RoboDK station: Sheet A.rdk

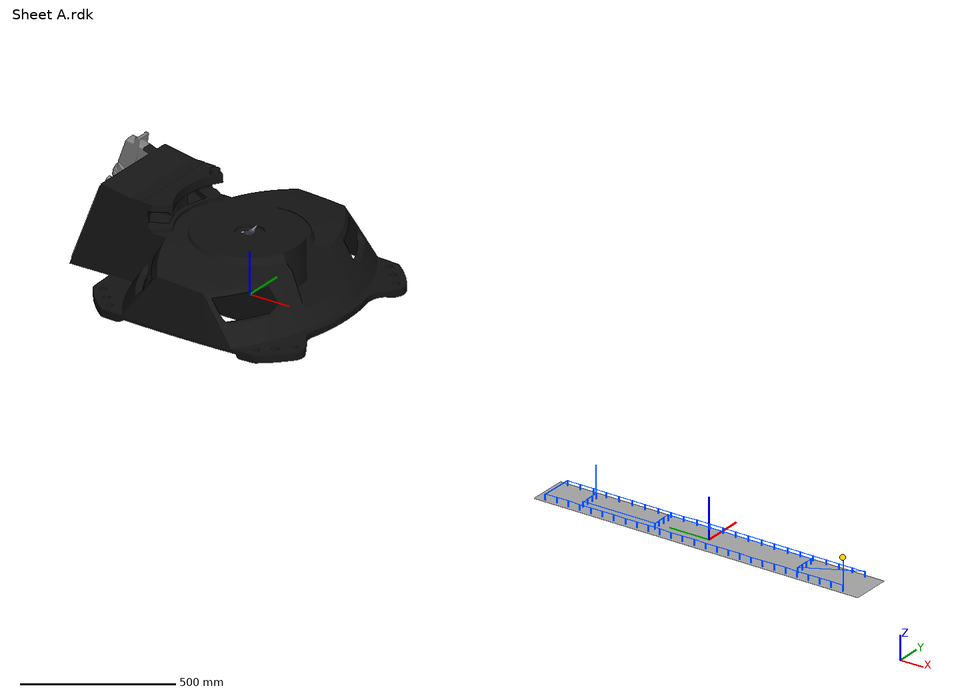
[picture v0: the station drawn from its stored meshes, robots at their saved joint values, targets as dots, program paths as lines]
Station Sheet A (saved by RoboDK 5.2.3). Poses are relative to the parent item; angles as X-Y-Z fixed-axis rotations.
  - frame KUKA KR 210 R2700 extra Base at (0, 0, 0) mm
    - robot KUKA KR 210 R2700 extra: 6 axes, payload 210 kg, reach 2696 mm, repeatability 0.06 mm, weight 1068 kg
        joint limits [-185, -140, -120, -350, -125, -350] to [185, -5, 155, 350, 125, 350]; home [0, -90, 90, 0, 0, 0]; saved at [-1.926, -24.263, 90.653, -184.563, 15.421, 182.902]
      - tool Spindle, TCP at (32, 0, 260) mm, rotated rx 0 ry 39 rz 0 deg, size 157.3 x 72 x 259.9 mm
  - frame Frame 2 at (1800, 0, -372.68) mm, rotated rx 0 ry 0 rz 90 deg
    - object Sheet A stp at (0, 0, 0) mm, size 148.8 x 1269.1 x 0.8 mm, geometry from Sheet A stp.stp
    - object Sheet A-box 1 Hole positioning at (0, 0, 0) mm, 63 curves, geometry from Point 63
  - machining project Point settings: rotZ(0) | rotX(0)*rotY(0) | rotZ(0) | onStart | onPathStart | onApproach | onPoint | onRetract | onFinish | SetRPM(%1) | SetTool(%1) | Extruder(%1) | default | default | OutOnMov(%1) | OutOffMov(%1) | onPathFinish | M_RunCode(%1)
  - program Point (326 instructions, listed below)
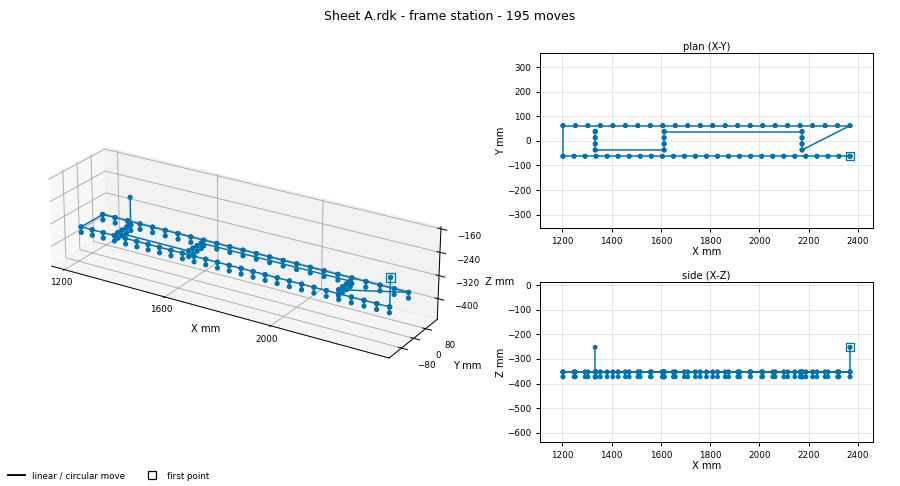
[picture p0: tool path of Sheet A.rdk in frame station, 195 of 195 moves have a stored position in this frame; points joined in program order, loops and branches not executed]

--- program Point (robot KUKA KR 210 R2700 extra) ---
  Smooth(1)
  Set speed (1000.0 mm/s)
  Set Ref.: Frame 2
  Set Tool: Spindle
  Show Spindle
  MoveJ 1 to (-62.4, -567.96, 120) mm, rotated rx -180 ry 0 rz 70 deg; joints [-0.851, -22.431, 74.95, -271.587, 12.949, 255.14]
  MoveL 2 to (-62.4, -567.96, 120) mm, rotated rx -180 ry 0 rz 70 deg; joints [-0.851, -22.431, 74.95, -271.587, 12.949, 255.14]
  MoveL 3 to (-62.4, -567.96, 20) mm, rotated rx 180 ry 0 rz 90 deg; joints [1.707, -18.651, 73.621, -164.804, 4.101, 166.168]
  MoveL 4 to (-62.4, -567.96, 20) mm, rotated rx 180 ry 0 rz 90 deg; joints [1.707, -18.651, 73.621, -164.804, 4.101, 166.168]
  Set speed (50.0 mm/s)
  MoveL 5 to (-62.4, -567.96, 0) mm, rotated rx 180 ry 0 rz 90 deg; joints [1.707, -17.786, 73.065, -165.856, 4.4, 167.222]
  MoveL 6 to (-62.4, -567.96, 20) mm, rotated rx 180 ry 0 rz 90 deg; joints [1.707, -18.651, 73.621, -164.804, 4.101, 166.168]
  Set speed (1000.0 mm/s)
  MoveL 7 to (-62.4, -523.11, 20) mm, rotated rx 180 ry 0 rz 90 deg; joints [1.744, -19.865, 76.907, -169.661, 6.127, 171.075]
  Set speed (50.0 mm/s)
  MoveL 8 to (-62.4, -523.11, 0) mm, rotated rx -180 ry 0 rz 90 deg; joints [1.744, -18.993, 76.358, -170.176, 6.446, 171.593]
  MoveL 9 to (-62.4, -523.11, 20) mm, rotated rx 180 ry 0 rz 90 deg; joints [1.744, -19.865, 76.907, -169.661, 6.127, 171.075]
  Set speed (1000.0 mm/s)
  MoveL 10 to (-62.4, -478.27, 20) mm, rotated rx -180 ry 0 rz 90 deg; joints [1.783, -20.997, 80.071, -172.048, 8.138, 173.513]
  Set speed (50.0 mm/s)
  MoveL 11 to (-62.4, -478.27, 0) mm, rotated rx 180 ry 0 rz 90 deg; joints [1.783, -20.115, 79.528, -172.362, 8.473, 173.831]
  MoveL 12 to (-62.4, -478.27, 20) mm, rotated rx -180 ry 0 rz 90 deg; joints [1.783, -20.997, 80.071, -172.048, 8.138, 173.513]
  Set speed (1000.0 mm/s)
  MoveL 13 to (-62.4, -433.42, 20) mm, rotated rx -180 ry 0 rz 90 deg; joints [1.824, -22.051, 83.128, -173.458, 10.127, 174.977]
  Set speed (50.0 mm/s)
  MoveL 14 to (-62.4, -433.42, 0) mm, rotated rx -180 ry 0 rz 90 deg; joints [1.824, -21.158, 82.588, -173.676, 10.478, 175.198]
  MoveL 15 to (-62.4, -433.42, 20) mm, rotated rx -180 ry 0 rz 90 deg; joints [1.824, -22.051, 83.128, -173.458, 10.127, 174.977]
  Set speed (1000.0 mm/s)
  MoveL 16 to (-62.4, -388.57, 20) mm, rotated rx -180 ry 0 rz 90 deg; joints [1.867, -23.031, 86.087, -174.386, 12.097, 175.961]
  Set speed (50.0 mm/s)
  MoveL 17 to (-62.4, -388.57, 0) mm, rotated rx -180 ry 0 rz 90 deg; joints [1.867, -22.126, 85.549, -174.549, 12.462, 176.127]
  MoveL 18 to (-62.4, -388.57, 20) mm, rotated rx -180 ry 0 rz 90 deg; joints [1.867, -23.031, 86.087, -174.386, 12.097, 175.961]
  Set speed (1000.0 mm/s)
  MoveL 19 to (-62.4, -343.73, 20) mm, rotated rx 180 ry 0 rz 90 deg; joints [1.912, -23.94, 88.957, -175.04, 14.053, 176.674]
  Set speed (50.0 mm/s)
  MoveL 20 to (-62.4, -343.73, 0) mm, rotated rx -180 ry 0 rz 90 deg; joints [1.912, -23.021, 88.419, -175.168, 14.431, 176.806]
  MoveL 21 to (-62.4, -343.73, 20) mm, rotated rx 180 ry 0 rz 90 deg; joints [1.912, -23.94, 88.957, -175.04, 14.053, 176.674]
  Set speed (1000.0 mm/s)
  MoveL 22 to (-62.4, -298.88, 20) mm, rotated rx -180 ry 0 rz 90 deg; joints [1.958, -24.779, 91.747, -175.524, 15.998, 177.219]
  Set speed (50.0 mm/s)
  MoveL 23 to (-62.4, -298.88, 0) mm, rotated rx -180 ry 0 rz 90 deg; joints [1.958, -23.846, 91.208, -175.629, 16.39, 177.328]
  MoveL 24 to (-62.4, -298.88, 20) mm, rotated rx -180 ry 0 rz 90 deg; joints [1.958, -24.779, 91.747, -175.524, 15.998, 177.219]
  Set speed (1000.0 mm/s)
  MoveL 25 to (-62.4, -254.03, 20) mm, rotated rx 180 ry 0 rz 90 deg; joints [2.008, -25.549, 94.461, -175.895, 17.937, 177.654]
  Set speed (50.0 mm/s)
  MoveL 26 to (-62.4, -254.03, 0) mm, rotated rx -180 ry 0 rz 90 deg; joints [2.008, -24.601, 93.92, -175.983, 18.343, 177.747]
  MoveL 27 to (-62.4, -254.03, 20) mm, rotated rx 180 ry 0 rz 90 deg; joints [2.008, -25.549, 94.461, -175.895, 17.937, 177.654]
  Set speed (1000.0 mm/s)
  MoveL 28 to (-62.4, -209.19, 20) mm, rotated rx 180 ry 0 rz 90 deg; joints [2.06, -26.252, 97.104, -176.185, 19.875, 178.013]
  Set speed (50.0 mm/s)
  MoveL 29 to (-62.4, -209.19, 0) mm, rotated rx 180 ry 0 rz 90 deg; joints [2.06, -25.287, 96.56, -176.261, 20.294, 178.093]
  MoveL 30 to (-62.4, -209.19, 20) mm, rotated rx 180 ry 0 rz 90 deg; joints [2.06, -26.252, 97.104, -176.185, 19.875, 178.013]
  Set speed (1000.0 mm/s)
  MoveL 31 to (-62.4, -164.34, 20) mm, rotated rx -180 ry 0 rz 90 deg; joints [2.114, -26.886, 99.683, -176.418, 21.817, 178.318]
  Set speed (50.0 mm/s)
  MoveL 32 to (-62.4, -164.34, 0) mm, rotated rx -180 ry 0 rz 90 deg; joints [2.114, -25.904, 99.134, -176.485, 22.249, 178.389]
  MoveL 33 to (-62.4, -164.34, 20) mm, rotated rx -180 ry 0 rz 90 deg; joints [2.114, -26.886, 99.683, -176.418, 21.817, 178.318]
  Set speed (1000.0 mm/s)
  MoveL 34 to (-62.4, -119.5, 20) mm, rotated rx -180 ry 0 rz 90 deg; joints [2.172, -27.45, 102.199, -176.607, 23.766, 178.583]
  Set speed (50.0 mm/s)
  MoveL 35 to (-62.4, -119.5, 0) mm, rotated rx 180 ry 0 rz 90 deg; joints [2.172, -26.45, 101.645, -176.666, 24.211, 178.647]
  MoveL 36 to (-62.4, -119.5, 20) mm, rotated rx -180 ry 0 rz 90 deg; joints [2.172, -27.45, 102.199, -176.607, 23.766, 178.583]
  Set speed (1000.0 mm/s)
  MoveL 37 to (-62.4, -74.65, 20) mm, rotated rx -180 ry 0 rz 90 deg; joints [2.233, -27.944, 104.657, -176.762, 25.728, 178.818]
  Set speed (50.0 mm/s)
  MoveL 38 to (-62.4, -74.65, 0) mm, rotated rx 180 ry 0 rz 90 deg; joints [2.233, -26.925, 104.096, -176.815, 26.185, 178.877]
  MoveL 39 to (-62.4, -74.65, 20) mm, rotated rx -180 ry 0 rz 90 deg; joints [2.233, -27.944, 104.657, -176.762, 25.728, 178.818]
  Set speed (1000.0 mm/s)
  MoveL 40 to (-62.4, -29.8, 20) mm, rotated rx 180 ry 0 rz 90 deg; joints [2.297, -28.365, 107.059, -176.89, 27.706, 179.032]
  Set speed (50.0 mm/s)
  MoveL 41 to (-62.4, -29.8, 0) mm, rotated rx 180 ry 0 rz 90 deg; joints [2.297, -27.326, 106.49, -176.938, 28.176, 179.086]
  MoveL 42 to (-62.4, -29.8, 20) mm, rotated rx 180 ry 0 rz 90 deg; joints [2.297, -28.365, 107.059, -176.89, 27.706, 179.032]
  Set speed (1000.0 mm/s)
  MoveL 43 to (-62.4, 15.04, 20) mm, rotated rx 180 ry 0 rz 90 deg; joints [2.365, -28.71, 109.405, -176.996, 29.705, 179.229]
  Set speed (50.0 mm/s)
  MoveL 44 to (-62.4, 15.04, 0) mm, rotated rx -180 ry 0 rz 90 deg; joints [2.365, -27.651, 108.829, -177.04, 30.187, 179.279]
  MoveL 45 to (-62.4, 15.04, 20) mm, rotated rx 180 ry 0 rz 90 deg; joints [2.365, -28.71, 109.405, -176.996, 29.705, 179.229]
  Set speed (1000.0 mm/s)
  MoveL 46 to (-62.4, 59.89, 20) mm, rotated rx 180 ry 0 rz 90 deg; joints [2.437, -28.977, 111.699, -177.083, 31.73, 179.413]
  Set speed (50.0 mm/s)
  MoveL 47 to (-62.4, 59.89, 0) mm, rotated rx 180 ry 0 rz 90 deg; joints [2.437, -27.896, 111.113, -177.123, 32.225, 179.46]
  MoveL 48 to (-62.4, 59.89, 20) mm, rotated rx 180 ry 0 rz 90 deg; joints [2.437, -28.977, 111.699, -177.083, 31.73, 179.413]
  Set speed (1000.0 mm/s)
  MoveL 49 to (-62.4, 104.73, 20) mm, rotated rx 180 ry 0 rz 90 deg; joints [2.514, -29.161, 113.941, -177.155, 33.786, 179.589]
  Set speed (50.0 mm/s)
  MoveL 50 to (-62.4, 104.73, 0) mm, rotated rx -180 ry 0 rz 90 deg; joints [2.514, -28.058, 113.345, -177.192, 34.292, 179.633]
  MoveL 51 to (-62.4, 104.73, 20) mm, rotated rx 180 ry 0 rz 90 deg; joints [2.514, -29.161, 113.941, -177.155, 33.786, 179.589]
  Set speed (1000.0 mm/s)
  MoveL 52 to (-62.4, 149.58, 20) mm, rotated rx -180 ry 0 rz 90 deg; joints [2.596, -29.258, 116.133, -177.212, 35.878, 179.759]
  Set speed (50.0 mm/s)
  MoveL 53 to (-62.4, 149.58, 0) mm, rotated rx -180 ry 0 rz 90 deg; joints [2.596, -28.132, 115.524, -177.247, 36.396, 179.801]
  MoveL 54 to (-62.4, 149.58, 20) mm, rotated rx -180 ry 0 rz 90 deg; joints [2.596, -29.258, 116.133, -177.212, 35.878, 179.759]
  Set speed (1000.0 mm/s)
  MoveL 55 to (-62.4, 194.43, 20) mm, rotated rx 180 ry 0 rz 90 deg; joints [2.683, -29.262, 118.273, -177.258, 38.012, 179.925]
  Set speed (50.0 mm/s)
  MoveL 56 to (-62.4, 194.43, 0) mm, rotated rx -180 ry 0 rz 90 deg; joints [2.683, -28.113, 117.652, -177.29, 38.54, 179.965]
  MoveL 57 to (-62.4, 194.43, 20) mm, rotated rx 180 ry 0 rz 90 deg; joints [2.683, -29.262, 118.273, -177.258, 38.012, 179.925]
  Set speed (1000.0 mm/s)
  MoveL 58 to (-62.4, 239.27, 20) mm, rotated rx 180 ry 0 rz 90 deg; joints [2.777, -29.169, 120.362, -177.293, 40.192, 180.09]
  Set speed (50.0 mm/s)
  MoveL 59 to (-62.4, 239.27, 0) mm, rotated rx 180 ry 0 rz 90 deg; joints [2.777, -27.996, 119.727, -177.322, 40.73, 180.129]
  MoveL 60 to (-62.4, 239.27, 20) mm, rotated rx 180 ry 0 rz 90 deg; joints [2.777, -29.169, 120.362, -177.293, 40.192, 180.09]
  Set speed (1000.0 mm/s)
  MoveL 61 to (-62.4, 284.12, 20) mm, rotated rx -180 ry 0 rz 90 deg; joints [2.877, -28.97, 122.4, -177.317, 42.426, 180.255]
  Set speed (50.0 mm/s)
  MoveL 62 to (-62.4, 284.12, 0) mm, rotated rx 180 ry 0 rz 90 deg; joints [2.877, -27.773, 121.75, -177.344, 42.973, 180.293]
  MoveL 63 to (-62.4, 284.12, 20) mm, rotated rx -180 ry 0 rz 90 deg; joints [2.877, -28.97, 122.4, -177.317, 42.426, 180.255]
  Set speed (1000.0 mm/s)
  MoveL 64 to (-62.4, 328.97, 20) mm, rotated rx 180 ry 0 rz 90 deg; joints [2.984, -28.658, 124.384, -177.331, 44.719, 180.423]
  Set speed (50.0 mm/s)
  MoveL 65 to (-62.4, 328.97, 0) mm, rotated rx 180 ry 0 rz 90 deg; joints [2.984, -27.438, 123.719, -177.357, 45.273, 180.459]
  MoveL 66 to (-62.4, 328.97, 20) mm, rotated rx 180 ry 0 rz 90 deg; joints [2.984, -28.658, 124.384, -177.331, 44.719, 180.423]
  Set speed (1000.0 mm/s)
  MoveL 67 to (-62.4, 373.81, 20) mm, rotated rx 180 ry 0 rz 90 deg; joints [3.1, -28.226, 126.314, -177.336, 47.078, 180.595]
  Set speed (50.0 mm/s)
  MoveL 68 to (-62.4, 373.81, 0) mm, rotated rx -180 ry 0 rz 90 deg; joints [3.1, -26.983, 125.632, -177.36, 47.638, 180.631]
  MoveL 69 to (-62.4, 373.81, 20) mm, rotated rx 180 ry 0 rz 90 deg; joints [3.1, -28.226, 126.314, -177.336, 47.078, 180.595]
  Set speed (1000.0 mm/s)
  MoveL 70 to (-62.4, 418.66, 20) mm, rotated rx 180 ry 0 rz 90 deg; joints [3.225, -27.664, 128.188, -177.331, 49.511, 180.774]
  Set speed (50.0 mm/s)
  MoveL 71 to (-62.4, 418.66, 0) mm, rotated rx 180 ry 0 rz 90 deg; joints [3.225, -26.399, 127.488, -177.354, 50.075, 180.809]
  MoveL 72 to (-62.4, 418.66, 20) mm, rotated rx 180 ry 0 rz 90 deg; joints [3.225, -27.664, 128.188, -177.331, 49.511, 180.774]
  Set speed (1000.0 mm/s)
  MoveL 73 to (-62.4, 463.5, 20) mm, rotated rx 180 ry 0 rz 90 deg; joints [3.361, -26.961, 130.003, -177.317, 52.024, 180.962]
  Set speed (50.0 mm/s)
  MoveL 74 to (-62.4, 463.5, 0) mm, rotated rx 180 ry 0 rz 90 deg; joints [3.361, -25.676, 129.284, -177.337, 52.589, 180.995]
  MoveL 75 to (-62.4, 463.5, 20) mm, rotated rx 180 ry 0 rz 90 deg; joints [3.361, -26.961, 130.003, -177.317, 52.024, 180.962]
  Set speed (1000.0 mm/s)
  MoveL 76 to (-62.4, 508.35, 20) mm, rotated rx 180 ry 0 rz 90 deg; joints [3.509, -26.107, 131.756, -177.292, 54.626, 181.16]
  Set speed (50.0 mm/s)
  MoveL 77 to (-62.4, 508.35, 0) mm, rotated rx 180 ry 0 rz 90 deg; joints [3.509, -24.803, 131.016, -177.311, 55.19, 181.193]
  MoveL 78 to (-62.4, 508.35, 20) mm, rotated rx 180 ry 0 rz 90 deg; joints [3.509, -26.107, 131.756, -177.292, 54.626, 181.16]
  Set speed (1000.0 mm/s)
  MoveL 79 to (-62.4, 553.2, 20) mm, rotated rx 180 ry 0 rz 90 deg; joints [3.67, -25.091, 133.443, -177.257, 57.325, 181.372]
  Set speed (50.0 mm/s)
  MoveL 80 to (-62.4, 553.2, 0) mm, rotated rx 180 ry 0 rz 90 deg; joints [3.67, -23.771, 132.682, -177.274, 57.882, 181.404]
  MoveL 81 to (-62.4, 553.2, 20) mm, rotated rx 180 ry 0 rz 90 deg; joints [3.67, -25.091, 133.443, -177.257, 57.325, 181.372]
  Set speed (1000.0 mm/s)
  MoveL 82 to (-62.4, 598.04, 20) mm, rotated rx 180 ry 0 rz 90 deg; joints [3.847, -23.899, 135.059, -177.209, 60.126, 181.601]
  Set speed (50.0 mm/s)
  MoveL 83 to (-62.4, 598.04, 0) mm, rotated rx 180 ry 0 rz 90 deg; joints [3.847, -22.567, 134.275, -177.224, 60.674, 181.631]
  MoveL 84 to (-62.4, 598.04, 20) mm, rotated rx 180 ry 0 rz 90 deg; joints [3.847, -23.899, 135.059, -177.209, 60.126, 181.601]
  Set speed (1000.0 mm/s)
  MoveL 85 to (61.9, 598.04, 20) mm, rotated rx 180 ry 0 rz 90 deg; joints [-3.817, -23.898, 135.06, -182.769, 60.129, 178.412]
  Set speed (50.0 mm/s)
  MoveL 86 to (61.9, 598.04, 0) mm, rotated rx -180 ry 0 rz 90 deg; joints [-3.817, -22.566, 134.277, -182.754, 60.676, 178.382]
  MoveL 87 to (61.9, 598.04, 20) mm, rotated rx 180 ry 0 rz 90 deg; joints [-3.817, -23.898, 135.06, -182.769, 60.129, 178.412]
  Set speed (1000.0 mm/s)
  MoveL 88 to (61.9, 547.35, 20) mm, rotated rx -180 ry 0 rz 90 deg; joints [-3.619, -25.232, 133.228, -182.716, 56.969, 178.667]
  Set speed (50.0 mm/s)
  MoveL 89 to (61.9, 547.35, 0) mm, rotated rx 180 ry 0 rz 90 deg; joints [-3.619, -23.914, 132.469, -182.699, 57.528, 178.636]
  MoveL 90 to (61.9, 547.35, 20) mm, rotated rx -180 ry 0 rz 90 deg; joints [-3.619, -25.232, 133.228, -182.716, 56.969, 178.667]
  Set speed (1000.0 mm/s)
  MoveL 91 to (61.9, 496.65, 20) mm, rotated rx -180 ry 0 rz 90 deg; joints [-3.442, -26.345, 131.306, -182.678, 53.941, 178.902]
  Set speed (50.0 mm/s)
  MoveL 92 to (61.9, 496.65, 0) mm, rotated rx 180 ry 0 rz 90 deg; joints [-3.442, -25.045, 130.572, -182.66, 54.505, 178.869]
  MoveL 93 to (61.9, 496.65, 20) mm, rotated rx -180 ry 0 rz 90 deg; joints [-3.442, -26.345, 131.306, -182.678, 53.941, 178.902]
  Set speed (1000.0 mm/s)
  MoveL 94 to (61.9, 445.96, 20) mm, rotated rx 180 ry 0 rz 90 deg; joints [-3.28, -27.253, 129.302, -182.655, 51.033, 179.12]
  Set speed (50.0 mm/s)
  MoveL 95 to (61.9, 445.96, 0) mm, rotated rx -180 ry 0 rz 90 deg; joints [-3.28, -25.975, 128.59, -182.634, 51.598, 179.086]
  MoveL 96 to (61.9, 445.96, 20) mm, rotated rx 180 ry 0 rz 90 deg; joints [-3.28, -27.253, 129.302, -182.655, 51.033, 179.12]
  Set speed (1000.0 mm/s)
  MoveL 97 to (61.9, 395.26, 20) mm, rotated rx -180 ry 0 rz 90 deg; joints [-3.134, -27.974, 127.219, -182.644, 48.234, 179.325]
  Set speed (50.0 mm/s)
  MoveL 98 to (61.9, 395.26, 0) mm, rotated rx 180 ry 0 rz 90 deg; joints [-3.134, -26.72, 126.528, -182.621, 48.796, 179.291]
  MoveL 99 to (61.9, 395.26, 20) mm, rotated rx -180 ry 0 rz 90 deg; joints [-3.134, -27.974, 127.219, -182.644, 48.234, 179.325]
  Set speed (1000.0 mm/s)
  MoveL 100 to (61.9, 344.56, 20) mm, rotated rx -180 ry 0 rz 90 deg; joints [-2.999, -28.522, 125.063, -182.645, 45.533, 179.521]
  Set speed (50.0 mm/s)
  MoveL 101 to (61.9, 344.56, 0) mm, rotated rx 180 ry 0 rz 90 deg; joints [-2.999, -27.294, 124.392, -182.62, 46.089, 179.486]
  MoveL 102 to (61.9, 344.56, 20) mm, rotated rx -180 ry 0 rz 90 deg; joints [-2.999, -28.522, 125.063, -182.645, 45.533, 179.521]
  Set speed (1000.0 mm/s)
  MoveL 103 to (61.9, 293.87, 20) mm, rotated rx 180 ry 0 rz 90 deg; joints [-2.876, -28.912, 122.837, -182.658, 42.92, 179.711]
  Set speed (50.0 mm/s)
  MoveL 104 to (61.9, 293.87, 0) mm, rotated rx 180 ry 0 rz 90 deg; joints [-2.876, -27.71, 122.184, -182.631, 43.469, 179.674]
  MoveL 105 to (61.9, 293.87, 20) mm, rotated rx 180 ry 0 rz 90 deg; joints [-2.876, -28.912, 122.837, -182.658, 42.92, 179.711]
  Set speed (1000.0 mm/s)
  MoveL 106 to (61.9, 243.17, 20) mm, rotated rx 180 ry 0 rz 90 deg; joints [-2.763, -29.155, 120.542, -182.683, 40.385, 179.897]
  Set speed (50.0 mm/s)
  MoveL 107 to (61.9, 243.17, 0) mm, rotated rx -180 ry 0 rz 90 deg; joints [-2.763, -27.98, 119.907, -182.654, 40.924, 179.858]
  MoveL 108 to (61.9, 243.17, 20) mm, rotated rx 180 ry 0 rz 90 deg; joints [-2.763, -29.155, 120.542, -182.683, 40.385, 179.897]
  Set speed (1000.0 mm/s)
  MoveL 109 to (61.9, 192.48, 20) mm, rotated rx 180 ry 0 rz 90 deg; joints [-2.658, -29.264, 118.182, -182.722, 37.919, 180.082]
  Set speed (50.0 mm/s)
  MoveL 110 to (61.9, 192.48, 0) mm, rotated rx 180 ry 0 rz 90 deg; joints [-2.658, -28.116, 117.562, -182.69, 38.447, 180.041]
  MoveL 111 to (61.9, 192.48, 20) mm, rotated rx 180 ry 0 rz 90 deg; joints [-2.658, -29.264, 118.182, -182.722, 37.919, 180.082]
  Set speed (1000.0 mm/s)
  MoveL 112 to (61.9, 141.78, 20) mm, rotated rx -180 ry 0 rz 90 deg; joints [-2.561, -29.248, 115.756, -182.774, 35.513, 180.268]
  Set speed (50.0 mm/s)
  MoveL 113 to (61.9, 141.78, 0) mm, rotated rx 180 ry 0 rz 90 deg; joints [-2.561, -28.125, 115.15, -182.74, 36.028, 180.226]
  MoveL 114 to (61.9, 141.78, 20) mm, rotated rx -180 ry 0 rz 90 deg; joints [-2.561, -29.248, 115.756, -182.774, 35.513, 180.268]
  Set speed (1000.0 mm/s)
  MoveL 115 to (61.9, 91.09, 20) mm, rotated rx 180 ry 0 rz 90 deg; joints [-2.47, -29.114, 113.266, -182.843, 33.158, 180.46]
  Set speed (50.0 mm/s)
  MoveL 116 to (61.9, 91.09, 0) mm, rotated rx 180 ry 0 rz 90 deg; joints [-2.47, -28.018, 112.673, -182.805, 33.661, 180.415]
  MoveL 117 to (61.9, 91.09, 20) mm, rotated rx 180 ry 0 rz 90 deg; joints [-2.47, -29.114, 113.266, -182.843, 33.158, 180.46]
  Set speed (1000.0 mm/s)
  MoveL 118 to (61.9, 40.39, 20) mm, rotated rx 180 ry 0 rz 90 deg; joints [-2.386, -28.871, 110.709, -182.929, 30.847, 180.66]
  Set speed (50.0 mm/s)
  MoveL 119 to (61.9, 40.39, 0) mm, rotated rx -180 ry 0 rz 90 deg; joints [-2.386, -27.799, 110.127, -182.888, 31.336, 180.612]
  MoveL 120 to (61.9, 40.39, 20) mm, rotated rx 180 ry 0 rz 90 deg; joints [-2.386, -28.871, 110.709, -182.929, 30.847, 180.66]
  Set speed (1000.0 mm/s)
  MoveL 121 to (61.9, -10.31, 20) mm, rotated rx 180 ry 0 rz 90 deg; joints [-2.307, -28.525, 108.086, -183.037, 28.573, 180.874]
  Set speed (50.0 mm/s)
  MoveL 122 to (61.9, -10.31, 0) mm, rotated rx -180 ry 0 rz 90 deg; joints [-2.307, -27.477, 107.514, -182.991, 29.048, 180.822]
  MoveL 123 to (61.9, -10.31, 20) mm, rotated rx 180 ry 0 rz 90 deg; joints [-2.307, -28.525, 108.086, -183.037, 28.573, 180.874]
  Set speed (1000.0 mm/s)
  MoveL 124 to (61.9, -61, 20) mm, rotated rx 180 ry 0 rz 90 deg; joints [-2.234, -28.08, 105.395, -183.17, 26.328, 181.106]
  Set speed (50.0 mm/s)
  MoveL 125 to (61.9, -61, 0) mm, rotated rx -180 ry 0 rz 90 deg; joints [-2.234, -27.055, 104.832, -183.12, 26.79, 181.049]
  MoveL 126 to (61.9, -61, 20) mm, rotated rx 180 ry 0 rz 90 deg; joints [-2.234, -28.08, 105.395, -183.17, 26.328, 181.106]
  Set speed (1000.0 mm/s)
  MoveL 127 to (61.9, -111.7, 20) mm, rotated rx 180 ry 0 rz 90 deg; joints [-2.165, -27.542, 102.632, -183.336, 24.107, 181.363]
  Set speed (50.0 mm/s)
  MoveL 128 to (61.9, -111.7, 0) mm, rotated rx 180 ry 0 rz 90 deg; joints [-2.165, -26.538, 102.077, -183.279, 24.554, 181.301]
  MoveL 129 to (61.9, -111.7, 20) mm, rotated rx 180 ry 0 rz 90 deg; joints [-2.165, -27.542, 102.632, -183.336, 24.107, 181.363]
  Set speed (1000.0 mm/s)
  MoveL 130 to (61.9, -162.39, 20) mm, rotated rx 180 ry 0 rz 90 deg; joints [-2.1, -26.912, 99.795, -183.544, 21.902, 181.657]
  Set speed (50.0 mm/s)
  MoveL 131 to (61.9, -162.39, 0) mm, rotated rx 180 ry 0 rz 90 deg; joints [-2.1, -25.93, 99.246, -183.479, 22.334, 181.586]
  MoveL 132 to (61.9, -162.39, 20) mm, rotated rx 180 ry 0 rz 90 deg; joints [-2.1, -26.912, 99.795, -183.544, 21.902, 181.657]
  Set speed (1000.0 mm/s)
  MoveL 133 to (61.9, -213.09, 20) mm, rotated rx 180 ry 0 rz 90 deg; joints [-2.039, -26.194, 96.878, -183.806, 19.707, 182]
  Set speed (50.0 mm/s)
  MoveL 134 to (61.9, -213.09, 0) mm, rotated rx 180 ry 0 rz 90 deg; joints [-2.039, -25.231, 96.334, -183.731, 20.125, 181.919]
  MoveL 135 to (61.9, -213.09, 20) mm, rotated rx 180 ry 0 rz 90 deg; joints [-2.039, -26.194, 96.878, -183.806, 19.707, 182]
  Set speed (1000.0 mm/s)
  MoveL 136 to (61.9, -263.78, 20) mm, rotated rx -180 ry 0 rz 90 deg; joints [-1.981, -25.388, 93.878, -184.145, 17.516, 182.413]
  Set speed (50.0 mm/s)
  MoveL 137 to (61.9, -263.78, 0) mm, rotated rx 180 ry 0 rz 90 deg; joints [-1.981, -24.443, 93.337, -184.054, 17.919, 182.319]
  MoveL 138 to (61.9, -263.78, 20) mm, rotated rx -180 ry 0 rz 90 deg; joints [-1.981, -25.388, 93.878, -184.145, 17.516, 182.413]
  Set speed (1000.0 mm/s)
  MoveL 139 to (61.9, -314.48, 20) mm, rotated rx -180 ry 0 rz 90 deg; joints [-1.926, -24.495, 90.786, -184.592, 15.322, 182.932]
  Set speed (50.0 mm/s)
  MoveL 140 to (61.9, -314.48, 0) mm, rotated rx -180 ry 0 rz 90 deg; joints [-1.926, -23.567, 90.248, -184.481, 15.71, 182.817]
  MoveL 141 to (61.9, -314.48, 20) mm, rotated rx -180 ry 0 rz 90 deg; joints [-1.926, -24.495, 90.786, -184.592, 15.322, 182.932]
  Set speed (1000.0 mm/s)
  MoveL 142 to (61.9, -365.18, 20) mm, rotated rx 180 ry 0 rz 90 deg; joints [-1.875, -23.514, 87.596, -185.204, 13.119, 183.612]
  Set speed (50.0 mm/s)
  MoveL 143 to (61.9, -365.18, 0) mm, rotated rx 180 ry 0 rz 90 deg; joints [-1.875, -22.602, 87.058, -185.063, 13.491, 183.467]
  MoveL 144 to (61.9, -365.18, 20) mm, rotated rx 180 ry 0 rz 90 deg; joints [-1.875, -23.514, 87.596, -185.204, 13.119, 183.612]
  Set speed (1000.0 mm/s)
  MoveL 145 to (61.9, -415.87, 20) mm, rotated rx -180 ry 0 rz 90 deg; joints [-1.826, -22.444, 84.298, -186.087, 10.9, 184.559]
  Set speed (50.0 mm/s)
  MoveL 146 to (61.9, -415.87, 0) mm, rotated rx -180 ry 0 rz 90 deg; joints [-1.826, -21.546, 83.759, -185.896, 11.257, 184.364]
  MoveL 147 to (61.9, -415.87, 20) mm, rotated rx -180 ry 0 rz 90 deg; joints [-1.826, -22.444, 84.298, -186.087, 10.9, 184.559]
  Set speed (1000.0 mm/s)
  MoveL 148 to (61.9, -466.57, 20) mm, rotated rx 180 ry 0 rz 90 deg; joints [-1.779, -21.28, 80.88, -187.458, 8.658, 185.991]
  Set speed (50.0 mm/s)
  MoveL 149 to (61.9, -466.57, 0) mm, rotated rx -180 ry 0 rz 90 deg; joints [-1.779, -20.395, 80.337, -187.178, 8.998, 185.707]
  MoveL 150 to (61.9, -466.57, 20) mm, rotated rx 180 ry 0 rz 90 deg; joints [-1.779, -21.28, 80.88, -187.458, 8.658, 185.991]
  Set speed (1000.0 mm/s)
  MoveL 151 to (61.9, -517.26, 20) mm, rotated rx -180 ry 0 rz 90 deg; joints [-1.735, -20.018, 77.328, -189.859, 6.39, 188.45]
  Set speed (50.0 mm/s)
  MoveL 152 to (61.9, -517.26, 0) mm, rotated rx 180 ry 0 rz 90 deg; joints [-1.735, -19.144, 76.779, -189.385, 6.711, 187.973]
  MoveL 153 to (61.9, -517.26, 20) mm, rotated rx -180 ry 0 rz 90 deg; joints [-1.735, -20.018, 77.328, -189.859, 6.39, 188.45]
  Set speed (1000.0 mm/s)
  MoveL 154 to (61.9, -567.96, 20) mm, rotated rx 180 ry 0 rz 90 deg; joints [-1.693, -18.651, 73.622, -195.076, 4.1, 193.723]
  Set speed (50.0 mm/s)
  MoveL 155 to (61.9, -567.96, 0) mm, rotated rx 180 ry 0 rz 90 deg; joints [-1.693, -17.786, 73.066, -194.033, 4.398, 192.677]
  MoveL 156 to (61.9, -567.96, 20) mm, rotated rx 180 ry 0 rz 90 deg; joints [-1.693, -18.651, 73.622, -195.076, 4.1, 193.723]
  Set speed (1000.0 mm/s)
  MoveL 157 to (-37, -372.96, 20) mm, rotated rx 180 ry 0 rz 90 deg; joints [1.116, -23.369, 87.139, -176.824, 12.783, 177.77]
  Set speed (50.0 mm/s)
  MoveL 158 to (-37, -372.96, 0) mm, rotated rx 180 ry 0 rz 90 deg; joints [1.116, -22.459, 86.601, -176.912, 13.154, 177.86]
  MoveL 159 to (-37, -372.96, 20) mm, rotated rx 180 ry 0 rz 90 deg; joints [1.116, -23.369, 87.139, -176.824, 12.783, 177.77]
  Set speed (1000.0 mm/s)
  MoveL 160 to (-12, -372.96, 20) mm, rotated rx 180 ry 0 rz 90 deg; joints [0.362, -23.376, 87.16, -178.97, 12.785, 179.277]
  Set speed (50.0 mm/s)
  MoveL 161 to (-12, -372.96, 0) mm, rotated rx 180 ry 0 rz 90 deg; joints [0.362, -22.466, 86.621, -178.999, 13.157, 179.307]
  MoveL 162 to (-12, -372.96, 20) mm, rotated rx 180 ry 0 rz 90 deg; joints [0.362, -23.376, 87.16, -178.97, 12.785, 179.277]
  Set speed (1000.0 mm/s)
  MoveL 163 to (13, -372.96, 20) mm, rotated rx -180 ry 0 rz 90 deg; joints [-0.392, -23.376, 87.159, -181.116, 12.785, 180.783]
  Set speed (50.0 mm/s)
  MoveL 164 to (13, -372.96, 0) mm, rotated rx -180 ry 0 rz 90 deg; joints [-0.392, -22.466, 86.621, -181.085, 13.157, 180.751]
  MoveL 165 to (13, -372.96, 20) mm, rotated rx -180 ry 0 rz 90 deg; joints [-0.392, -23.376, 87.159, -181.116, 12.785, 180.783]
  Set speed (1000.0 mm/s)
  MoveL 166 to (38, -372.96, 20) mm, rotated rx -180 ry 0 rz 90 deg; joints [-1.146, -23.369, 87.138, -183.262, 12.783, 182.291]
  Set speed (50.0 mm/s)
  MoveL 167 to (38, -372.96, 0) mm, rotated rx 180 ry 0 rz 90 deg; joints [-1.146, -22.459, 86.599, -183.172, 13.154, 182.198]
  MoveL 168 to (38, -372.96, 20) mm, rotated rx -180 ry 0 rz 90 deg; joints [-1.146, -23.369, 87.138, -183.262, 12.783, 182.291]
  Set speed (1000.0 mm/s)
  MoveL 169 to (38, 187.04, 20) mm, rotated rx 180 ry 0 rz 90 deg; joints [-1.626, -29.268, 117.967, -181.673, 37.7, 180.06]
  Set speed (50.0 mm/s)
  MoveL 170 to (38, 187.04, 0) mm, rotated rx 180 ry 0 rz 90 deg; joints [-1.626, -28.122, 117.348, -181.653, 38.227, 180.035]
  MoveL 171 to (38, 187.04, 20) mm, rotated rx 180 ry 0 rz 90 deg; joints [-1.626, -29.268, 117.967, -181.673, 37.7, 180.06]
  Set speed (1000.0 mm/s)
  MoveL 172 to (13, 187.04, 20) mm, rotated rx 180 ry 0 rz 90 deg; joints [-0.556, -29.267, 117.99, -180.572, 37.723, 180.02]
  Set speed (50.0 mm/s)
  MoveL 173 to (13, 187.04, 0) mm, rotated rx 180 ry 0 rz 90 deg; joints [-0.556, -28.121, 117.371, -180.565, 38.25, 180.012]
  MoveL 174 to (13, 187.04, 20) mm, rotated rx 180 ry 0 rz 90 deg; joints [-0.556, -29.267, 117.99, -180.572, 37.723, 180.02]
  Set speed (1000.0 mm/s)
  MoveL 175 to (-12, 187.04, 20) mm, rotated rx -180 ry 0 rz 90 deg; joints [0.514, -29.267, 117.99, -179.472, 37.723, 179.981]
  Set speed (50.0 mm/s)
  MoveL 176 to (-12, 187.04, 0) mm, rotated rx -180 ry 0 rz 90 deg; joints [0.514, -28.121, 117.371, -179.478, 38.25, 179.989]
  MoveL 177 to (-12, 187.04, 20) mm, rotated rx -180 ry 0 rz 90 deg; joints [0.514, -29.267, 117.99, -179.472, 37.723, 179.981]
  Set speed (1000.0 mm/s)
  MoveL 178 to (-37, 187.04, 20) mm, rotated rx 180 ry 0 rz 90 deg; joints [1.583, -29.268, 117.969, -178.371, 37.701, 179.941]
  Set speed (50.0 mm/s)
  MoveL 179 to (-37, 187.04, 0) mm, rotated rx 180 ry 0 rz 90 deg; joints [1.583, -28.122, 117.35, -178.39, 38.228, 179.966]
  MoveL 180 to (-37, 187.04, 20) mm, rotated rx 180 ry 0 rz 90 deg; joints [1.583, -29.268, 117.969, -178.371, 37.701, 179.941]
  Set speed (1000.0 mm/s)
  MoveL 181 to (-37, 467.04, 20) mm, rotated rx 180 ry 0 rz 90 deg; joints [2.001, -26.878, 130.191, -178.409, 52.306, 180.582]
  Set speed (50.0 mm/s)
  MoveL 182 to (-37, 467.04, 0) mm, rotated rx 180 ry 0 rz 90 deg; joints [2.001, -25.591, 129.469, -178.421, 52.872, 180.602]
  MoveL 183 to (-37, 467.04, 20) mm, rotated rx 180 ry 0 rz 90 deg; joints [2.001, -26.878, 130.191, -178.409, 52.306, 180.582]
  Set speed (1000.0 mm/s)
  MoveL 184 to (-12, 467.04, 20) mm, rotated rx 180 ry 0 rz 90 deg; joints [0.649, -26.868, 130.214, -179.484, 52.345, 180.189]
  Set speed (50.0 mm/s)
  MoveL 185 to (-12, 467.04, 0) mm, rotated rx 180 ry 0 rz 90 deg; joints [0.649, -25.58, 129.492, -179.488, 52.911, 180.196]
  MoveL 186 to (-12, 467.04, 20) mm, rotated rx 180 ry 0 rz 90 deg; joints [0.649, -26.868, 130.214, -179.484, 52.345, 180.189]
  Set speed (1000.0 mm/s)
  MoveL 187 to (13, 467.04, 20) mm, rotated rx 180 ry 0 rz 90 deg; joints [-0.703, -26.868, 130.214, -180.559, 52.344, 179.795]
  Set speed (50.0 mm/s)
  MoveL 188 to (13, 467.04, 0) mm, rotated rx 180 ry 0 rz 90 deg; joints [-0.703, -25.581, 129.492, -180.555, 52.91, 179.788]
  MoveL 189 to (13, 467.04, 20) mm, rotated rx 180 ry 0 rz 90 deg; joints [-0.703, -26.868, 130.214, -180.559, 52.344, 179.795]
  Set speed (1000.0 mm/s)
  MoveL 190 to (38, 467.04, 20) mm, rotated rx 180 ry 0 rz 90 deg; joints [-2.055, -26.879, 130.19, -181.634, 52.304, 179.402]
  Set speed (50.0 mm/s)
  MoveL 191 to (38, 467.04, 0) mm, rotated rx 180 ry 0 rz 90 deg; joints [-2.055, -25.592, 129.468, -181.622, 52.869, 179.382]
  MoveL 192 to (38, 467.04, 20) mm, rotated rx 180 ry 0 rz 90 deg; joints [-2.055, -26.879, 130.19, -181.634, 52.304, 179.402]
  MoveL 193 to (38, 467.04, 20) mm, rotated rx 180 ry 0 rz 90 deg; joints [-2.055, -26.879, 130.19, -181.634, 52.304, 179.402]
  Set speed (1000.0 mm/s)
  MoveL 194 to (38, 467.04, 20) mm, rotated rx 180 ry 0 rz 90 deg; joints [-2.055, -26.879, 130.19, -181.634, 52.304, 179.402]
  MoveL 195 to (38, 467.04, 120) mm, rotated rx 180 ry 0 rz 90 deg; joints [-2.055, -33.597, 133.575, -181.714, 48.973, 179.528]
